ABB RAPID module: 00A6084E

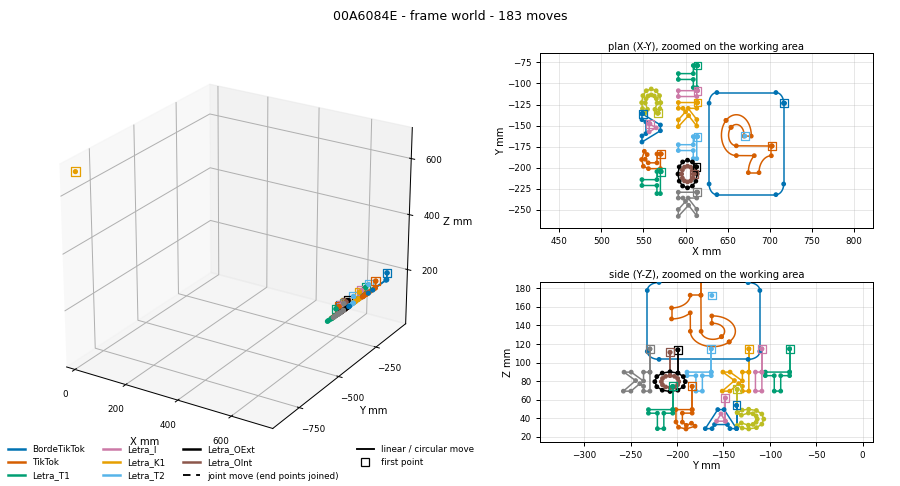
[picture p0: tool path of 00A6084E in frame world, 183 of 183 moves have a stored position in this frame; points joined in program order, loops and branches not executed]
MODULE Module1
        CONST robtarget Target_130_BordeTikTokInicio:=[[92.878,251.287,20],[0.27059805,-0.653281482,0.653281482,0.27059805],[-1,0,-1,0],[9E+09,9E+09,9E+09,9E+09,9E+09,9E+09]];
    CONST robtarget Target_140:=[[83.933,247.582,20],[0.27059805,-0.653281482,0.653281482,0.27059805],[-1,0,-1,0],[9E+09,9E+09,9E+09,9E+09,9E+09,9E+09]];
    CONST robtarget Target_150:=[[80.227,238.636,20],[0.27059805,-0.653281482,0.653281482,0.27059805],[-1,0,-1,0],[9E+09,9E+09,9E+09,9E+09,9E+09,9E+09]];
    CONST robtarget Target_160:=[[80.227,142.704,20],[0.27059805,-0.653281482,0.653281482,0.27059805],[-1,0,-1,0],[9E+09,9E+09,9E+09,9E+09,9E+09,9E+09]];
    CONST robtarget Target_170:=[[83.933,133.759,20],[0.27059805,-0.653281482,0.653281482,0.27059805],[-1,0,-1,0],[9E+09,9E+09,9E+09,9E+09,9E+09,9E+09]];
    CONST robtarget Target_180:=[[92.878,130.054,20],[0.27059805,-0.653281482,0.653281482,0.27059805],[-1,0,-1,0],[9E+09,9E+09,9E+09,9E+09,9E+09,9E+09]];
    CONST robtarget Target_190:=[[188.81,130.054,20],[0.27059805,-0.653281482,0.653281482,0.27059805],[-1,0,-1,0],[9E+09,9E+09,9E+09,9E+09,9E+09,9E+09]];
    CONST robtarget Target_200:=[[197.755,133.759,20],[0.27059805,-0.653281482,0.653281482,0.27059805],[-1,0,-1,0],[9E+09,9E+09,9E+09,9E+09,9E+09,9E+09]];
    CONST robtarget Target_210:=[[201.46,142.704,20],[0.27059805,-0.653281482,0.653281482,0.27059805],[-1,0,-1,0],[9E+09,9E+09,9E+09,9E+09,9E+09,9E+09]];
    CONST robtarget Target_220:=[[201.46,238.636,20],[0.27059805,-0.653281482,0.653281482,0.27059805],[-1,0,-1,0],[9E+09,9E+09,9E+09,9E+09,9E+09,9E+09]];
    CONST robtarget Target_230:=[[197.755,247.582,20],[0.27059805,-0.653281482,0.653281482,0.27059805],[-1,0,-1,0],[9E+09,9E+09,9E+09,9E+09,9E+09,9E+09]];
    CONST robtarget Target_240_BordeTikTokFinal:=[[188.81,251.287,20],[0.27059805,-0.653281482,0.653281482,0.27059805],[-1,0,-1,0],[9E+09,9E+09,9E+09,9E+09,9E+09,9E+09]];
    CONST robtarget Target_250_TikTokInicio:=[[143.706205367,231.257091716,20.000126522],[0.27059805,-0.653281482,0.653281482,0.27059805],[0,0,0,0],[9E+09,9E+09,9E+09,9E+09,9E+09,9E+09]];
    CONST robtarget Target_260:=[[143.479220622,174.279999139,20.000159098],[0.27059805,-0.653281482,0.653281482,0.27059805],[0,0,0,0],[9E+09,9E+09,9E+09,9E+09,9E+09,9E+09]];
    CONST robtarget Target_270:=[[135.378239234,162.526330146,20.000165817],[0.27059805,-0.653281482,0.653281482,0.27059805],[0,0,0,0],[9E+09,9E+09,9E+09,9E+09,9E+09,9E+09]];
    CONST robtarget Target_280:=[[121.484474213,165.803207899,20.000163944],[0.27059805,-0.653281482,0.653281482,0.27059805],[0,0,0,0],[9E+09,9E+09,9E+09,9E+09,9E+09,9E+09]];
    CONST robtarget Target_290:=[[119.489363555,179.938064379,20.000155863],[0.27059805,-0.653281482,0.653281482,0.27059805],[0,0,0,0],[9E+09,9E+09,9E+09,9E+09,9E+09,9E+09]];
    CONST robtarget Target_300:=[[131.933354464,186.932471038,20.000151864],[0.27059805,-0.653281482,0.653281482,0.27059805],[0,0,0,0],[9E+09,9E+09,9E+09,9E+09,9E+09,9E+09]];
    CONST robtarget Target_310:=[[131.979634785,198.549631032,20.000145222],[0.27059805,-0.653281482,0.653281482,0.27059805],[0,0,0,0],[9E+09,9E+09,9E+09,9E+09,9E+09,9E+09]];
    CONST robtarget Target_320:=[[108.772618252,184.400845477,20.000153312],[0.27059805,-0.653281482,0.653281482,0.27059805],[0,0,0,0],[9E+09,9E+09,9E+09,9E+09,9E+09,9E+09]];
    CONST robtarget Target_330:=[[113.281741814,157.597458494,20.000168635],[0.27059805,-0.653281482,0.653281482,0.27059805],[0,0,0,0],[9E+09,9E+09,9E+09,9E+09,9E+09,9E+09]];
    CONST robtarget Target_340:=[[139.840807855,151.820802015,20.000171938],[0.27059805,-0.653281482,0.653281482,0.27059805],[0,0,0,0],[9E+09,9E+09,9E+09,9E+09,9E+09,9E+09]];
    CONST robtarget Target_350:=[[155.075499923,174.329864782,20.000159069],[0.27059805,-0.653281482,0.653281482,0.27059805],[0,0,0,0],[9E+09,9E+09,9E+09,9E+09,9E+09,9E+09]];
    CONST robtarget Target_360:=[[155.17372753,203.510585817,20.000142385],[0.27059805,-0.653281482,0.653281482,0.27059805],[0,0,0,0],[9E+09,9E+09,9E+09,9E+09,9E+09,9E+09]];
    CONST robtarget Target_370:=[[167.73702862,194.971199808,20.000147268],[0.27059805,-0.653281482,0.653281482,0.27059805],[0,0,0,0],[9E+09,9E+09,9E+09,9E+09,9E+09,9E+09]];
    CONST robtarget Target_380:=[[175.332383248,193.829143916,20.000147921],[0.27059805,-0.653281482,0.653281482,0.27059805],[0,0,0,0],[9E+09,9E+09,9E+09,9E+09,9E+09,9E+09]];
    CONST robtarget Target_390:=[[175.332383248,211.188020458,20.000137996],[0.27059805,-0.653281482,0.653281482,0.27059805],[0,0,0,0],[9E+09,9E+09,9E+09,9E+09,9E+09,9E+09]];
    CONST robtarget Target_400:=[[161.14267515,217.065945812,20.00013646],[0.27059805,-0.653281482,0.653281482,0.27059805],[0,0,0,0],[9E+09,9E+09,9E+09,9E+09,9E+09,9E+09]];
    CONST robtarget Target_410_TikTokFinal:=[[155.26722819,231.257091716,20.000126522],[0.27059805,-0.653281482,0.653281482,0.27059805],[0,0,0,0],[9E+09,9E+09,9E+09,9E+09,9E+09,9E+09]];
    CONST robtarget Target_415_T1Inicio:=[[48.177,110.059,20],[0.27059805,-0.653281482,0.653281482,0.27059805],[-1,1,-2,0],[9E+09,9E+09,9E+09,9E+09,9E+09,9E+09]];
    CONST robtarget Target_420:=[[48.174,104.402,20],[0.27059805,-0.653281482,0.653281482,0.27059805],[-1,1,-2,0],[9E+09,9E+09,9E+09,9E+09,9E+09,9E+09]];
    CONST robtarget Target_430:=[[57.774,104.396,20],[0.27059805,-0.653281482,0.653281482,0.27059805],[-1,1,-2,0],[9E+09,9E+09,9E+09,9E+09,9E+09,9E+09]];
    CONST robtarget Target_440:=[[57.759,80.053,20],[0.27059805,-0.653281482,0.653281482,0.27059805],[-1,1,-2,0],[9E+09,9E+09,9E+09,9E+09,9E+09,9E+09]];
    CONST robtarget Target_450:=[[64.701,80.049,20],[0.27059805,-0.653281482,0.653281482,0.27059805],[-1,1,-2,0],[9E+09,9E+09,9E+09,9E+09,9E+09,9E+09]];
    CONST robtarget Target_460:=[[64.717,104.392,20],[0.27059805,-0.653281482,0.653281482,0.27059805],[-1,1,-2,0],[9E+09,9E+09,9E+09,9E+09,9E+09,9E+09]];
    CONST robtarget Target_470:=[[74.317,104.386,20],[0.27059805,-0.653281482,0.653281482,0.27059805],[-1,1,-2,0],[9E+09,9E+09,9E+09,9E+09,9E+09,9E+09]];
    CONST robtarget Target_480_T1Final:=[[74.32,110.043,20],[0.27059805,-0.653281482,0.653281482,0.27059805],[-1,1,-2,0],[9E+09,9E+09,9E+09,9E+09,9E+09,9E+09]];
    CONST robtarget Target_490_IInicio:=[[78.049,110.041,20],[0.27059805,-0.653281482,0.653281482,0.27059805],[-1,1,-2,0],[9E+09,9E+09,9E+09,9E+09,9E+09,9E+09]];
    CONST robtarget Target_500:=[[78.03,80.041,20],[0.27059805,-0.653281482,0.653281482,0.27059805],[-1,1,-2,0],[9E+09,9E+09,9E+09,9E+09,9E+09,9E+09]];
    CONST robtarget Target_510:=[[84.973,80.036,20],[0.27059805,-0.653281482,0.653281482,0.27059805],[-1,1,-2,0],[9E+09,9E+09,9E+09,9E+09,9E+09,9E+09]];
    CONST robtarget Target_520_IFinal:=[[84.992,110.036,20],[0.27059805,-0.653281482,0.653281482,0.27059805],[-1,1,-2,0],[9E+09,9E+09,9E+09,9E+09,9E+09,9E+09]];
    CONST robtarget Target_530_K1Inicio:=[[92.106,110.032,20],[0.27059805,-0.653281482,0.653281482,0.27059805],[-1,1,-2,0],[9E+09,9E+09,9E+09,9E+09,9E+09,9E+09]];
    CONST robtarget Target_540:=[[92.087,80.032,20],[0.27059805,-0.653281482,0.653281482,0.27059805],[-1,1,-2,0],[9E+09,9E+09,9E+09,9E+09,9E+09,9E+09]];
    CONST robtarget Target_550:=[[98.987,80.028,20],[0.27059805,-0.653281482,0.653281482,0.27059805],[-1,1,-2,0],[9E+09,9E+09,9E+09,9E+09,9E+09,9E+09]];
    CONST robtarget Target_560:=[[98.992,87.613,20],[0.27059805,-0.653281482,0.653281482,0.27059805],[-1,1,-2,0],[9E+09,9E+09,9E+09,9E+09,9E+09,9E+09]];
    CONST robtarget Target_570:=[[103.023,91.811,20],[0.27059805,-0.653281482,0.653281482,0.27059805],[-1,1,-2,0],[9E+09,9E+09,9E+09,9E+09,9E+09,9E+09]];
    CONST robtarget Target_580:=[[112.616,80.019,20],[0.27059805,-0.653281482,0.653281482,0.27059805],[-1,1,-2,0],[9E+09,9E+09,9E+09,9E+09,9E+09,9E+09]];
    CONST robtarget Target_590:=[[120.716,80.014,20],[0.27059805,-0.653281482,0.653281482,0.27059805],[-1,1,-2,0],[9E+09,9E+09,9E+09,9E+09,9E+09,9E+09]];
    CONST robtarget Target_600:=[[107.569,96.651,20],[0.27059805,-0.653281482,0.653281482,0.27059805],[-1,1,-2,0],[9E+09,9E+09,9E+09,9E+09,9E+09,9E+09]];
    CONST robtarget Target_610:=[[120.006,110.015,20],[0.27059805,-0.653281482,0.653281482,0.27059805],[-1,0,-2,0],[9E+09,9E+09,9E+09,9E+09,9E+09,9E+09]];
    CONST robtarget Target_620:=[[112.292,110.019,20],[0.27059805,-0.653281482,0.653281482,0.27059805],[-1,1,-2,0],[9E+09,9E+09,9E+09,9E+09,9E+09,9E+09]];
    CONST robtarget Target_630:=[[98.997,96.013,20],[0.27059805,-0.653281482,0.653281482,0.27059805],[-1,1,-2,0],[9E+09,9E+09,9E+09,9E+09,9E+09,9E+09]];
    CONST robtarget Target_640_K1Final:=[[99.006,110.028,20],[0.27059805,-0.653281482,0.653281482,0.27059805],[-1,1,-2,0],[9E+09,9E+09,9E+09,9E+09,9E+09,9E+09]];
    CONST robtarget Target_650_T2Inicio:=[[132.563,110.007,20],[0.27059805,-0.653281482,0.653281482,0.27059805],[0,0,0,0],[9E+09,9E+09,9E+09,9E+09,9E+09,9E+09]];
    CONST robtarget Target_660:=[[132.559,104.35,20],[0.27059805,-0.653281482,0.653281482,0.27059805],[-1,1,-2,0],[9E+09,9E+09,9E+09,9E+09,9E+09,9E+09]];
    CONST robtarget Target_670:=[[142.159,104.344,20],[0.27059805,-0.653281482,0.653281482,0.27059805],[-1,0,-2,0],[9E+09,9E+09,9E+09,9E+09,9E+09,9E+09]];
    CONST robtarget Target_680:=[[142.144,80.001,20],[0.27059805,-0.653281482,0.653281482,0.27059805],[-1,1,-2,0],[9E+09,9E+09,9E+09,9E+09,9E+09,9E+09]];
    CONST robtarget Target_690:=[[149.087,79.996,20],[0.27059805,-0.653281482,0.653281482,0.27059805],[-1,1,-2,0],[9E+09,9E+09,9E+09,9E+09,9E+09,9E+09]];
    CONST robtarget Target_700:=[[149.102,104.339,20],[0.27059805,-0.653281482,0.653281482,0.27059805],[-1,0,-2,0],[9E+09,9E+09,9E+09,9E+09,9E+09,9E+09]];
    CONST robtarget Target_710:=[[158.702,104.333,20],[0.27059805,-0.653281482,0.653281482,0.27059805],[-1,0,-2,0],[9E+09,9E+09,9E+09,9E+09,9E+09,9E+09]];
    CONST robtarget Target_720_T2Final:=[[158.706,109.99,20],[0.27059805,-0.653281482,0.653281482,0.27059805],[-1,0,-2,0],[9E+09,9E+09,9E+09,9E+09,9E+09,9E+09]];
    CONST robtarget Target_730_OExtInicio:=[[168.541,108.484,20],[0.27059805,-0.653281482,0.653281482,0.27059805],[0,0,0,0],[9E+09,9E+09,9E+09,9E+09,9E+09,9E+09]];
    CONST robtarget Target_740:=[[162.666,102.938,20],[0.27059805,-0.653281482,0.653281482,0.27059805],[-1,0,-2,0],[9E+09,9E+09,9E+09,9E+09,9E+09,9E+09]];
    CONST robtarget Target_750:=[[160.539,94.989,20],[0.27059805,-0.653281482,0.653281482,0.27059805],[-1,1,-2,0],[9E+09,9E+09,9E+09,9E+09,9E+09,9E+09]];
    CONST robtarget Target_760:=[[162.656,87.038,20],[0.27059805,-0.653281482,0.653281482,0.27059805],[-1,1,-2,0],[9E+09,9E+09,9E+09,9E+09,9E+09,9E+09]];
    CONST robtarget Target_770:=[[168.524,81.484,20],[0.27059805,-0.653281482,0.653281482,0.27059805],[-1,1,-2,0],[9E+09,9E+09,9E+09,9E+09,9E+09,9E+09]];
    CONST robtarget Target_780:=[[176.944,79.465,20],[0.27059805,-0.653281482,0.653281482,0.27059805],[-1,1,-2,0],[9E+09,9E+09,9E+09,9E+09,9E+09,9E+09]];
    CONST robtarget Target_790:=[[185.345,81.474,20],[0.27059805,-0.653281482,0.653281482,0.27059805],[-1,1,-2,0],[9E+09,9E+09,9E+09,9E+09,9E+09,9E+09]];
    CONST robtarget Target_800:=[[191.22,87.02,20],[0.27059805,-0.653281482,0.653281482,0.27059805],[-1,0,-2,0],[9E+09,9E+09,9E+09,9E+09,9E+09,9E+09]];
    CONST robtarget Target_810:=[[193.368,94.969,20],[0.27059805,-0.653281482,0.653281482,0.27059805],[-1,0,-2,0],[9E+09,9E+09,9E+09,9E+09,9E+09,9E+09]];
    CONST robtarget Target_820:=[[191.23,102.92,20],[0.27059805,-0.653281482,0.653281482,0.27059805],[-1,0,-2,0],[9E+09,9E+09,9E+09,9E+09,9E+09,9E+09]];
    CONST robtarget Target_830:=[[185.362,108.474,20],[0.27059805,-0.653281482,0.653281482,0.27059805],[-1,0,-2,0],[9E+09,9E+09,9E+09,9E+09,9E+09,9E+09]];
    CONST robtarget Target_840_OExtFinal:=[[176.963,110.493,20],[0.27059805,-0.653281482,0.653281482,0.27059805],[-1,0,-2,0],[9E+09,9E+09,9E+09,9E+09,9E+09,9E+09]];
    CONST robtarget Target_850_OIntInicio:=[[176.96,104.579,20],[0.27059805,-0.653281482,0.653281482,0.27059805],[0,0,0,0],[9E+09,9E+09,9E+09,9E+09,9E+09,9E+09]];
    CONST robtarget Target_860:=[[172.159,103.361,20],[0.27059805,-0.653281482,0.653281482,0.27059805],[-1,0,-2,0],[9E+09,9E+09,9E+09,9E+09,9E+09,9E+09]];
    CONST robtarget Target_870:=[[168.792,99.956,20],[0.27059805,-0.653281482,0.653281482,0.27059805],[-1,0,-2,0],[9E+09,9E+09,9E+09,9E+09,9E+09,9E+09]];
    CONST robtarget Target_880:=[[167.568,94.985,20],[0.27059805,-0.653281482,0.653281482,0.27059805],[-1,0,-2,0],[9E+09,9E+09,9E+09,9E+09,9E+09,9E+09]];
    CONST robtarget Target_890:=[[168.786,90.013,20],[0.27059805,-0.653281482,0.653281482,0.27059805],[-1,1,-2,0],[9E+09,9E+09,9E+09,9E+09,9E+09,9E+09]];
    CONST robtarget Target_900:=[[172.148,86.603,20],[0.27059805,-0.653281482,0.653281482,0.27059805],[-1,1,-2,0],[9E+09,9E+09,9E+09,9E+09,9E+09,9E+09]];
    CONST robtarget Target_910:=[[176.948,85.379,20],[0.27059805,-0.653281482,0.653281482,0.27059805],[-1,1,-2,0],[9E+09,9E+09,9E+09,9E+09,9E+09,9E+09]];
    CONST robtarget Target_920:=[[181.748,86.597,20],[0.27059805,-0.653281482,0.653281482,0.27059805],[-1,1,-2,0],[9E+09,9E+09,9E+09,9E+09,9E+09,9E+09]];
    CONST robtarget Target_930:=[[185.115,90.003,20],[0.27059805,-0.653281482,0.653281482,0.27059805],[-1,0,-2,0],[9E+09,9E+09,9E+09,9E+09,9E+09,9E+09]];
    CONST robtarget Target_940:=[[186.339,94.973,20],[0.27059805,-0.653281482,0.653281482,0.27059805],[-1,0,-2,0],[9E+09,9E+09,9E+09,9E+09,9E+09,9E+09]];
    CONST robtarget Target_950:=[[185.121,99.945,20],[0.27059805,-0.653281482,0.653281482,0.27059805],[-1,0,-2,0],[9E+09,9E+09,9E+09,9E+09,9E+09,9E+09]];
    CONST robtarget Target_960_OIntFinal:=[[181.759,103.355,20],[0.27059805,-0.653281482,0.653281482,0.27059805],[-1,0,-2,0],[9E+09,9E+09,9E+09,9E+09,9E+09,9E+09]];
    CONST robtarget Target_970_K2Inicio:=[[198.606,109.966,20],[0.27059805,-0.653281482,0.653281482,0.27059805],[0,0,0,0],[9E+09,9E+09,9E+09,9E+09,9E+09,9E+09]];
    CONST robtarget Target_980:=[[198.587,79.966,20],[0.27059805,-0.653281482,0.653281482,0.27059805],[-1,1,-2,0],[9E+09,9E+09,9E+09,9E+09,9E+09,9E+09]];
    CONST robtarget Target_990:=[[205.487,79.961,20],[0.27059805,-0.653281482,0.653281482,0.27059805],[-1,0,-2,0],[9E+09,9E+09,9E+09,9E+09,9E+09,9E+09]];
    CONST robtarget Target_1000:=[[205.492,87.547,20],[0.27059805,-0.653281482,0.653281482,0.27059805],[-1,0,-2,0],[9E+09,9E+09,9E+09,9E+09,9E+09,9E+09]];
    CONST robtarget Target_1010:=[[209.523,91.744,20],[0.27059805,-0.653281482,0.653281482,0.27059805],[-1,0,-2,0],[9E+09,9E+09,9E+09,9E+09,9E+09,9E+09]];
    CONST robtarget Target_1020:=[[219.116,79.953,20],[0.27059805,-0.653281482,0.653281482,0.27059805],[-1,0,-2,0],[9E+09,9E+09,9E+09,9E+09,9E+09,9E+09]];
    CONST robtarget Target_1030:=[[227.216,79.948,20],[0.27059805,-0.653281482,0.653281482,0.27059805],[-1,0,-2,0],[9E+09,9E+09,9E+09,9E+09,9E+09,9E+09]];
    CONST robtarget Target_1040:=[[214.069,96.584,20],[0.27059805,-0.653281482,0.653281482,0.27059805],[-1,0,-2,0],[9E+09,9E+09,9E+09,9E+09,9E+09,9E+09]];
    CONST robtarget Target_1050:=[[226.506,109.948,20],[0.27059805,-0.653281482,0.653281482,0.27059805],[-1,0,-1,0],[9E+09,9E+09,9E+09,9E+09,9E+09,9E+09]];
    CONST robtarget Target_1060:=[[218.792,109.953,20],[0.27059805,-0.653281482,0.653281482,0.27059805],[-1,0,-2,0],[9E+09,9E+09,9E+09,9E+09,9E+09,9E+09]];
    CONST robtarget Target_1070:=[[205.497,95.947,20],[0.27059805,-0.653281482,0.653281482,0.27059805],[-1,0,-2,0],[9E+09,9E+09,9E+09,9E+09,9E+09,9E+09]];
    CONST robtarget Target_1080_K2Final:=[[205.506,109.961,20],[0.27059805,-0.653281482,0.653281482,0.27059805],[-1,0,-2,0],[9E+09,9E+09,9E+09,9E+09,9E+09,9E+09]];
    CONST robtarget Target_1090_CInicio:=[[104.623,46.124,20],[0.27059805,-0.653281482,0.653281482,0.27059805],[-1,1,-2,0],[9E+09,9E+09,9E+09,9E+09,9E+09,9E+09]];
    CONST robtarget Target_1100:=[[99.333,50.07,20],[0.27059805,-0.653281482,0.653281482,0.27059805],[-1,1,-2,0],[9E+09,9E+09,9E+09,9E+09,9E+09,9E+09]];
    CONST robtarget Target_1110:=[[92.284,51.446,20],[0.27059805,-0.653281482,0.653281482,0.27059805],[-1,1,-2,0],[9E+09,9E+09,9E+09,9E+09,9E+09,9E+09]];
    CONST robtarget Target_1120:=[[83.947,49.459,20],[0.27059805,-0.653281482,0.653281482,0.27059805],[-1,1,-2,0],[9E+09,9E+09,9E+09,9E+09,9E+09,9E+09]];
    CONST robtarget Target_1130:=[[78.115,43.934,20],[0.27059805,-0.653281482,0.653281482,0.27059805],[-1,1,-2,0],[9E+09,9E+09,9E+09,9E+09,9E+09,9E+09]];
    CONST robtarget Target_1140:=[[75.988,35.942,20],[0.27059805,-0.653281482,0.653281482,0.27059805],[-1,1,-2,0],[9E+09,9E+09,9E+09,9E+09,9E+09,9E+09]];
    CONST robtarget Target_1150:=[[78.105,27.948,20],[0.27059805,-0.653281482,0.653281482,0.27059805],[-1,1,-2,0],[9E+09,9E+09,9E+09,9E+09,9E+09,9E+09]];
    CONST robtarget Target_1160:=[[83.93,22.416,20],[0.27059805,-0.653281482,0.653281482,0.27059805],[-1,1,-2,0],[9E+09,9E+09,9E+09,9E+09,9E+09,9E+09]];
    CONST robtarget Target_1170:=[[92.221,20.418,20],[0.27059805,-0.653281482,0.653281482,0.27059805],[-1,1,-2,0],[9E+09,9E+09,9E+09,9E+09,9E+09,9E+09]];
    CONST robtarget Target_1180:=[[99.294,21.785,20],[0.27059805,-0.653281482,0.653281482,0.27059805],[-1,1,-2,0],[9E+09,9E+09,9E+09,9E+09,9E+09,9E+09]];
    CONST robtarget Target_1190:=[[104.61,25.767,20],[0.27059805,-0.653281482,0.653281482,0.27059805],[-1,1,-2,0],[9E+09,9E+09,9E+09,9E+09,9E+09,9E+09]];
    CONST robtarget Target_1200:=[[100.156,29.884,20],[0.27059805,-0.653281482,0.653281482,0.27059805],[-1,1,-2,0],[9E+09,9E+09,9E+09,9E+09,9E+09,9E+09]];
    CONST robtarget Target_1210:=[[92.611,26.332,20],[0.27059805,-0.653281482,0.653281482,0.27059805],[-1,1,-2,0],[9E+09,9E+09,9E+09,9E+09,9E+09,9E+09]];
    CONST robtarget Target_1220:=[[87.64,27.556,20],[0.27059805,-0.653281482,0.653281482,0.27059805],[-1,1,-2,0],[9E+09,9E+09,9E+09,9E+09,9E+09,9E+09]];
    CONST robtarget Target_1230:=[[84.235,30.965,20],[0.27059805,-0.653281482,0.653281482,0.27059805],[-1,1,-2,0],[9E+09,9E+09,9E+09,9E+09,9E+09,9E+09]];
    CONST robtarget Target_1240:=[[83.017,35.938,20],[0.27059805,-0.653281482,0.653281482,0.27059805],[-1,1,-2,0],[9E+09,9E+09,9E+09,9E+09,9E+09,9E+09]];
    CONST robtarget Target_1250:=[[84.241,40.908,20],[0.27059805,-0.653281482,0.653281482,0.27059805],[-1,1,-2,0],[9E+09,9E+09,9E+09,9E+09,9E+09,9E+09]];
    CONST robtarget Target_1260:=[[87.651,44.313,20],[0.27059805,-0.653281482,0.653281482,0.27059805],[-1,1,-2,0],[9E+09,9E+09,9E+09,9E+09,9E+09,9E+09]];
    CONST robtarget Target_1270:=[[92.623,45.532,20],[0.27059805,-0.653281482,0.653281482,0.27059805],[-1,1,-2,0],[9E+09,9E+09,9E+09,9E+09,9E+09,9E+09]];
    CONST robtarget Target_1280_CFinal:=[[100.163,42.013,20],[0.27059805,-0.653281482,0.653281482,0.27059805],[-1,1,-2,0],[9E+09,9E+09,9E+09,9E+09,9E+09,9E+09]];
    CONST robtarget Target_1290_AExtInicio:=[[105.336,20.924,20],[0.27059805,-0.653281482,0.653281482,0.27059805],[-1,1,-2,0],[9E+09,9E+09,9E+09,9E+09,9E+09,9E+09]];
    CONST robtarget Target_1300:=[[118.726,50.915,20],[0.27059805,-0.653281482,0.653281482,0.27059805],[-1,1,-2,0],[9E+09,9E+09,9E+09,9E+09,9E+09,9E+09]];
    CONST robtarget Target_1310:=[[125.583,50.911,20],[0.27059805,-0.653281482,0.653281482,0.27059805],[-1,1,-2,0],[9E+09,9E+09,9E+09,9E+09,9E+09,9E+09]];
    CONST robtarget Target_1320:=[[138.979,20.903,20],[0.27059805,-0.653281482,0.653281482,0.27059805],[-1,1,-2,0],[9E+09,9E+09,9E+09,9E+09,9E+09,9E+09]];
    CONST robtarget Target_1330:=[[131.693,20.907,20],[0.27059805,-0.653281482,0.653281482,0.27059805],[-1,1,-2,0],[9E+09,9E+09,9E+09,9E+09,9E+09,9E+09]];
    CONST robtarget Target_1340:=[[129.04,27.338,20],[0.27059805,-0.653281482,0.653281482,0.27059805],[-1,1,-2,0],[9E+09,9E+09,9E+09,9E+09,9E+09,9E+09]];
    CONST robtarget Target_1350:=[[115.111,27.346,20],[0.27059805,-0.653281482,0.653281482,0.27059805],[-1,1,-2,0],[9E+09,9E+09,9E+09,9E+09,9E+09,9E+09]];
    CONST robtarget Target_1360_AExtFinal:=[[112.45,20.919,20],[0.27059805,-0.653281482,0.653281482,0.27059805],[-1,1,-2,0],[9E+09,9E+09,9E+09,9E+09,9E+09,9E+09]];
    CONST robtarget Target_1400_JInicio:=[[153.14,50.894,20],[0.27059805,-0.653281482,0.653281482,0.27059805],[-1,1,-2,0],[9E+09,9E+09,9E+09,9E+09,9E+09,9E+09]];
    CONST robtarget Target_1410:=[[153.137,45.322,20],[0.27059805,-0.653281482,0.653281482,0.27059805],[-1,1,-2,0],[9E+09,9E+09,9E+09,9E+09,9E+09,9E+09]];
    CONST robtarget Target_1420:=[[163.68,45.316,20],[0.27059805,-0.653281482,0.653281482,0.27059805],[-1,1,-2,0],[9E+09,9E+09,9E+09,9E+09,9E+09,9E+09]];
    CONST robtarget Target_1430:=[[163.671,31.044,20],[0.27059805,-0.653281482,0.653281482,0.27059805],[-1,1,-2,0],[9E+09,9E+09,9E+09,9E+09,9E+09,9E+09]];
    CONST robtarget Target_1440:=[[159.425,26.076,20],[0.27059805,-0.653281482,0.653281482,0.27059805],[-1,1,-2,0],[9E+09,9E+09,9E+09,9E+09,9E+09,9E+09]];
    CONST robtarget Target_1450:=[[153.856,29.379,20],[0.27059805,-0.653281482,0.653281482,0.27059805],[-1,1,-2,0],[9E+09,9E+09,9E+09,9E+09,9E+09,9E+09]];
    CONST robtarget Target_1460:=[[149.996,24.753,20],[0.27059805,-0.653281482,0.653281482,0.27059805],[-1,1,-2,0],[9E+09,9E+09,9E+09,9E+09,9E+09,9E+09]];
    CONST robtarget Target_1470:=[[159.764,20.375,20],[0.27059805,-0.653281482,0.653281482,0.27059805],[-1,1,-2,0],[9E+09,9E+09,9E+09,9E+09,9E+09,9E+09]];
    CONST robtarget Target_1480:=[[167.823,23.135,20],[0.27059805,-0.653281482,0.653281482,0.27059805],[-1,1,-2,0],[9E+09,9E+09,9E+09,9E+09,9E+09,9E+09]];
    CONST robtarget Target_1490:=[[170.571,31.426,20],[0.27059805,-0.653281482,0.653281482,0.27059805],[-1,1,-2,0],[9E+09,9E+09,9E+09,9E+09,9E+09,9E+09]];
    CONST robtarget Target_1500_JFinal:=[[170.583,50.883,20],[0.27059805,-0.653281482,0.653281482,0.27059805],[-1,1,-2,0],[9E+09,9E+09,9E+09,9E+09,9E+09,9E+09]];
    CONST robtarget Target_1510_T3Inicio:=[[174.055,50.881,20],[0.27059805,-0.653281482,0.653281482,0.27059805],[-1,1,-2,0],[9E+09,9E+09,9E+09,9E+09,9E+09,9E+09]];
    CONST robtarget Target_1520:=[[174.051,45.224,20],[0.27059805,-0.653281482,0.653281482,0.27059805],[-1,1,-2,0],[9E+09,9E+09,9E+09,9E+09,9E+09,9E+09]];
    CONST robtarget Target_1530:=[[183.651,45.218,20],[0.27059805,-0.653281482,0.653281482,0.27059805],[-1,1,-2,0],[9E+09,9E+09,9E+09,9E+09,9E+09,9E+09]];
    CONST robtarget Target_1540:=[[183.636,20.875,20],[0.27059805,-0.653281482,0.653281482,0.27059805],[-1,1,-2,0],[9E+09,9E+09,9E+09,9E+09,9E+09,9E+09]];
    CONST robtarget Target_1550:=[[190.579,20.871,20],[0.27059805,-0.653281482,0.653281482,0.27059805],[-1,1,-2,0],[9E+09,9E+09,9E+09,9E+09,9E+09,9E+09]];
    CONST robtarget Target_1560:=[[190.594,45.213,20],[0.27059805,-0.653281482,0.653281482,0.27059805],[-1,1,-2,0],[9E+09,9E+09,9E+09,9E+09,9E+09,9E+09]];
    CONST robtarget Target_1570:=[[200.194,45.207,20],[0.27059805,-0.653281482,0.653281482,0.27059805],[-1,1,-2,0],[9E+09,9E+09,9E+09,9E+09,9E+09,9E+09]];
    CONST robtarget Target_1580_T3Final:=[[200.198,50.865,20],[0.27059805,-0.653281482,0.653281482,0.27059805],[-1,1,-2,0],[9E+09,9E+09,9E+09,9E+09,9E+09,9E+09]];
    CONST robtarget Target_1370_AIntInicio:=[[117.343,32.616,20],[0.27059805,-0.653281482,0.653281482,0.27059805],[-1,1,-2,0],[9E+09,9E+09,9E+09,9E+09,9E+09,9E+09]];
    CONST robtarget Target_1380:=[[122.108,44.099,20],[0.27059805,-0.653281482,0.653281482,0.27059805],[-1,1,-2,0],[9E+09,9E+09,9E+09,9E+09,9E+09,9E+09]];
    CONST robtarget Target_1390_AIntFinal:=[[126.858,32.61,20],[0.27059805,-0.653281482,0.653281482,0.27059805],[-1,1,-2,0],[9E+09,9E+09,9E+09,9E+09,9E+09,9E+09]];
    CONST robtarget Target_130_BordeTikTokInicio_4:=[[92.878,268.964669525,37.677669535],[0.27059805,-0.653281482,0.653281482,0.27059805],[-1,0,-1,0],[9E+09,9E+09,9E+09,9E+09,9E+09,9E+09]];
    CONST robtarget Target_250_TikTokInicio_2:=[[143.706205367,248.934761241,37.677796057],[0.27059805,-0.653281482,0.653281482,0.27059805],[-1,0,-1,0],[9E+09,9E+09,9E+09,9E+09,9E+09,9E+09]];
    CONST robtarget Target_415_T1Inicio_2:=[[48.177,127.736669525,37.677669535],[0.27059805,-0.653281482,0.653281482,0.27059805],[-1,0,-1,0],[9E+09,9E+09,9E+09,9E+09,9E+09,9E+09]];
    CONST robtarget Target_490_IInicio_2:=[[78.049,127.718669525,37.677669535],[0.27059805,-0.653281482,0.653281482,0.27059805],[-1,0,-1,0],[9E+09,9E+09,9E+09,9E+09,9E+09,9E+09]];
    CONST robtarget Target_530_K1Inicio_2:=[[92.106,127.709669525,37.677669535],[0.27059805,-0.653281482,0.653281482,0.27059805],[-1,0,-1,0],[9E+09,9E+09,9E+09,9E+09,9E+09,9E+09]];
    CONST robtarget Target_650_T2Inicio_2:=[[132.563,127.684669525,37.677669535],[0.27059805,-0.653281482,0.653281482,0.27059805],[-1,0,-1,0],[9E+09,9E+09,9E+09,9E+09,9E+09,9E+09]];
    CONST robtarget Target_730_OExtInicio_2:=[[168.541,126.161669525,37.677669535],[0.27059805,-0.653281482,0.653281482,0.27059805],[-1,0,-1,0],[9E+09,9E+09,9E+09,9E+09,9E+09,9E+09]];
    CONST robtarget Target_850_OIntInicio_3:=[[176.96,122.256669525,37.677669535],[0.27059805,-0.653281482,0.653281482,0.27059805],[-1,0,-1,0],[9E+09,9E+09,9E+09,9E+09,9E+09,9E+09]];
    CONST robtarget Target_970_K2Inicio_2:=[[198.606,127.643669525,37.677669535],[0.27059805,-0.653281482,0.653281482,0.27059805],[-1,0,-1,0],[9E+09,9E+09,9E+09,9E+09,9E+09,9E+09]];
    CONST robtarget Target_1090_CInicio_2:=[[104.623,63.801669525,37.677669535],[0.27059805,-0.653281482,0.653281482,0.27059805],[-1,1,-2,0],[9E+09,9E+09,9E+09,9E+09,9E+09,9E+09]];
    CONST robtarget Target_1290_AExtInicio_2:=[[105.336,38.601669525,37.677669535],[0.27059805,-0.653281482,0.653281482,0.27059805],[-1,1,-2,0],[9E+09,9E+09,9E+09,9E+09,9E+09,9E+09]];
    CONST robtarget Target_1400_JInicio_2:=[[153.14,68.571669525,37.677669535],[0.27059805,-0.653281482,0.653281482,0.27059805],[-1,1,-2,0],[9E+09,9E+09,9E+09,9E+09,9E+09,9E+09]];
    CONST robtarget Target_1510_T3Inicio_2:=[[174.055,68.558669525,37.677669535],[0.27059805,-0.653281482,0.653281482,0.27059805],[-1,1,-2,0],[9E+09,9E+09,9E+09,9E+09,9E+09,9E+09]];
    CONST robtarget Target_1370_AIntInicio_2:=[[117.343,50.293669525,37.677669535],[0.27059805,-0.653281482,0.653281482,0.27059805],[-1,1,-2,0],[9E+09,9E+09,9E+09,9E+09,9E+09,9E+09]];
    CONST robtarget PosMantenimiento:=[[842.764,64.247888054,868.878653416],[0.859297836,-0.339353237,0.355932818,-0.140564712],[-2,0,-1,0],[9E+09,9E+09,9E+09,9E+09,9E+09,9E+09]];
    PERS tooldata MyNewTool:=[TRUE,[[120.323,-0.111,166.727],[0.923879533,0,-0.382683432,0]],[1,[0,0,1],[1,0,0,0],0,0,0]];
    TASK PERS wobjdata Workobject_1:=[FALSE,TRUE,"",[[546.66,-30.515,0],[0.657678091,0.259729722,-0.259729722,-0.657678091]],[[0,0,0],[1,0,0,0]]];
    CONST robtarget MyHome:=[[131.933354464,208.145674467,41.213355305],[0.27059805,-0.653281482,0.653281482,0.27059805],[0,0,0,0],[9E+09,9E+09,9E+09,9E+09,9E+09,9E+09]];
!***********************************************************
    !
    ! M?dulo:  Module1
    !
    ! Descripción:
    !   <Introduzca la descripción aquí>
    !
    ! Autor: Cami
    !
    ! Versión: 1.0
    !
    !***********************************************************


    !***********************************************************
    !
    ! Procedimiento Main
    !
    !   Este es el punto de entrada de su programa
    !
    !***********************************************************
    PROC main()
        VAR bool mant := FALSE;

        WHILE TRUE DO

            IF DI_01 = 1 THEN
                SetDO DO_02,1;
                COMPLETO;
                SetDO DO_02,0;
            ENDIF

            IF DI_02 = 1 THEN
                IF mant = FALSE THEN
                    mant := TRUE;
                    Home;
                ELSE
                    mant := FALSE;
                    SetDO DO_02,1;
                    Mantenimiento;
                    SetDO DO_02,0;
                ENDIF

            ENDIF

        ENDWHILE
        SetDO DO_02,0;
        SetDO DO_02,1;
    ENDPROC
    PROC COMPLETO()
        BordeTikTok;
        TikTok;
        Letra_T1;
        Letra_I;
        Letra_K1;
        Letra_T2;
        Letra_OExt;
        Letra_OInt;
        Letra_K2;
        Letra_C;
        Letra_AExt;
        Letra_AInt;
        Letra_J;
        Letra_T3;
    ENDPROC
    PROC BordeTikTok()
        MoveJ Target_130_BordeTikTokInicio_4,v100,z100,MyNewTool\WObj:=Workobject_1;
        MoveJ Target_130_BordeTikTokInicio,v400,z100,MyNewTool\WObj:=Workobject_1;
        MoveC Target_140,Target_150,v100,z100,MyNewTool\WObj:=Workobject_1;
        MoveL Target_160,v100,z100,MyNewTool\WObj:=Workobject_1;
        MoveC Target_170,Target_180,v100,z100,MyNewTool\WObj:=Workobject_1;
        MoveL Target_190,v100,z100,MyNewTool\WObj:=Workobject_1;
        MoveC Target_200,Target_210,v100,z100,MyNewTool\WObj:=Workobject_1;
        MoveL Target_220,v100,z100,MyNewTool\WObj:=Workobject_1;
        MoveC Target_230,Target_240_BordeTikTokFinal,v100,z100,MyNewTool\WObj:=Workobject_1;
        MoveL Target_130_BordeTikTokInicio,v100,z100,MyNewTool\WObj:=Workobject_1;
        MoveL Target_130_BordeTikTokInicio_4,v100,z100,MyNewTool\WObj:=Workobject_1;
    ENDPROC
    PROC TikTok()
        MoveL Target_250_TikTokInicio_2,v100,z100,MyNewTool\WObj:=Workobject_1;
        MoveL Target_250_TikTokInicio,v100,z100,MyNewTool\WObj:=Workobject_1;
        MoveL Target_260,v100,z100,MyNewTool\WObj:=Workobject_1;
        MoveC Target_270,Target_280,v100,z100,MyNewTool\WObj:=Workobject_1;
        MoveL Target_280,v100,z100,MyNewTool\WObj:=Workobject_1;
        MoveC Target_290,Target_300,v100,z100,MyNewTool\WObj:=Workobject_1;
        MoveL Target_310,v100,z100,MyNewTool\WObj:=Workobject_1;
        MoveC Target_320,Target_330,v100,z100,MyNewTool\WObj:=Workobject_1;
        MoveL Target_330,v100,z100,MyNewTool\WObj:=Workobject_1;
        MoveC Target_340,Target_350,v100,z100,MyNewTool\WObj:=Workobject_1;
        MoveL Target_360,v100,z100,MyNewTool\WObj:=Workobject_1;
        MoveC Target_370,Target_380,v100,z100,MyNewTool\WObj:=Workobject_1;
        MoveL Target_390,v100,z100,MyNewTool\WObj:=Workobject_1;
        MoveC Target_400,Target_410_TikTokFinal,v100,z100,MyNewTool\WObj:=Workobject_1;
        MoveL Target_250_TikTokInicio,v100,z100,MyNewTool\WObj:=Workobject_1;
        MoveL Target_250_TikTokInicio_2,v100,z100,MyNewTool\WObj:=Workobject_1;
    ENDPROC
    PROC Letra_T1()
        MoveL Target_415_T1Inicio_2,v100,z100,MyNewTool\WObj:=Workobject_1;
        MoveL Target_415_T1Inicio,v100,z100,MyNewTool\WObj:=Workobject_1;
        MoveL Target_420,v100,z100,MyNewTool\WObj:=Workobject_1;
        MoveL Target_430,v100,z100,MyNewTool\WObj:=Workobject_1;
        MoveL Target_440,v100,z100,MyNewTool\WObj:=Workobject_1;
        MoveL Target_450,v100,z100,MyNewTool\WObj:=Workobject_1;
        MoveL Target_460,v100,z100,MyNewTool\WObj:=Workobject_1;
        MoveL Target_470,v100,z100,MyNewTool\WObj:=Workobject_1;
        MoveL Target_480_T1Final,v100,z100,MyNewTool\WObj:=Workobject_1;
        MoveL Target_415_T1Inicio,v100,z100,MyNewTool\WObj:=Workobject_1;
        MoveL Target_415_T1Inicio_2,v100,z100,MyNewTool\WObj:=Workobject_1;
    ENDPROC
    PROC Letra_I()
        MoveL Target_490_IInicio_2,v100,z100,MyNewTool\WObj:=Workobject_1;
        MoveL Target_490_IInicio,v100,z100,MyNewTool\WObj:=Workobject_1;
        MoveL Target_500,v100,z100,MyNewTool\WObj:=Workobject_1;
        MoveL Target_510,v100,z100,MyNewTool\WObj:=Workobject_1;
        MoveL Target_520_IFinal,v100,z100,MyNewTool\WObj:=Workobject_1;
        MoveL Target_490_IInicio,v100,z100,MyNewTool\WObj:=Workobject_1;
        MoveL Target_490_IInicio_2,v100,z100,MyNewTool\WObj:=Workobject_1;
    ENDPROC
    PROC Letra_K1()
        MoveL Target_530_K1Inicio_2,v100,z100,MyNewTool\WObj:=Workobject_1;
        MoveL Target_530_K1Inicio,v100,z100,MyNewTool\WObj:=Workobject_1;
        MoveL Target_540,v100,z100,MyNewTool\WObj:=Workobject_1;
        MoveL Target_550,v100,z100,MyNewTool\WObj:=Workobject_1;
        MoveL Target_560,v100,z100,MyNewTool\WObj:=Workobject_1;
        MoveL Target_570,v100,z100,MyNewTool\WObj:=Workobject_1;
        MoveL Target_580,v100,z100,MyNewTool\WObj:=Workobject_1;
        MoveL Target_590,v100,z100,MyNewTool\WObj:=Workobject_1;
        MoveL Target_600,v100,z100,MyNewTool\WObj:=Workobject_1;
        MoveL Target_610,v100,z100,MyNewTool\WObj:=Workobject_1;
        MoveL Target_620,v100,z100,MyNewTool\WObj:=Workobject_1;
        MoveL Target_630,v100,z100,MyNewTool\WObj:=Workobject_1;
        MoveL Target_640_K1Final,v100,z100,MyNewTool\WObj:=Workobject_1;
        MoveL Target_530_K1Inicio,v100,z100,MyNewTool\WObj:=Workobject_1;
        MoveL Target_530_K1Inicio_2,v100,z100,MyNewTool\WObj:=Workobject_1;
    ENDPROC
    PROC Letra_T2()
        MoveL Target_650_T2Inicio_2,v100,z100,MyNewTool\WObj:=Workobject_1;
        MoveL Target_650_T2Inicio,v100,z100,MyNewTool\WObj:=Workobject_1;
        MoveL Target_660,v100,z100,MyNewTool\WObj:=Workobject_1;
        MoveL Target_670,v100,z100,MyNewTool\WObj:=Workobject_1;
        MoveL Target_680,v100,z100,MyNewTool\WObj:=Workobject_1;
        MoveL Target_690,v100,z100,MyNewTool\WObj:=Workobject_1;
        MoveL Target_700,v100,z100,MyNewTool\WObj:=Workobject_1;
        MoveL Target_710,v100,z100,MyNewTool\WObj:=Workobject_1;
        MoveL Target_720_T2Final,v100,z100,MyNewTool\WObj:=Workobject_1;
        MoveL Target_650_T2Inicio,v100,z100,MyNewTool\WObj:=Workobject_1;
        MoveL Target_650_T2Inicio_2,v100,z100,MyNewTool\WObj:=Workobject_1;
    ENDPROC
    PROC Letra_OExt()
        MoveL Target_730_OExtInicio_2,v100,z100,MyNewTool\WObj:=Workobject_1;
        MoveL Target_730_OExtInicio,v100,z100,MyNewTool\WObj:=Workobject_1;
        MoveL Target_740,v100,z100,MyNewTool\WObj:=Workobject_1;
        MoveL Target_750,v100,z100,MyNewTool\WObj:=Workobject_1;
        MoveL Target_760,v100,z100,MyNewTool\WObj:=Workobject_1;
        MoveL Target_770,v100,z100,MyNewTool\WObj:=Workobject_1;
        MoveL Target_780,v100,z100,MyNewTool\WObj:=Workobject_1;
        MoveL Target_790,v100,z100,MyNewTool\WObj:=Workobject_1;
        MoveL Target_800,v100,z100,MyNewTool\WObj:=Workobject_1;
        MoveL Target_810,v100,z100,MyNewTool\WObj:=Workobject_1;
        MoveL Target_820,v100,z100,MyNewTool\WObj:=Workobject_1;
        MoveL Target_830,v100,z100,MyNewTool\WObj:=Workobject_1;
        MoveL Target_840_OExtFinal,v100,z100,MyNewTool\WObj:=Workobject_1;
        MoveL Target_730_OExtInicio,v100,z100,MyNewTool\WObj:=Workobject_1;
        MoveL Target_730_OExtInicio_2,v100,z100,MyNewTool\WObj:=Workobject_1;
    ENDPROC
    PROC Letra_OInt()
        MoveL Target_850_OIntInicio_3,v100,z100,MyNewTool\WObj:=Workobject_1;
        MoveL Target_850_OIntInicio,v100,z100,MyNewTool\WObj:=Workobject_1;
        MoveL Target_860,v100,z100,MyNewTool\WObj:=Workobject_1;
        MoveL Target_870,v100,z100,MyNewTool\WObj:=Workobject_1;
        MoveL Target_880,v100,z100,MyNewTool\WObj:=Workobject_1;
        MoveL Target_890,v100,z100,MyNewTool\WObj:=Workobject_1;
        MoveL Target_900,v100,z100,MyNewTool\WObj:=Workobject_1;
        MoveL Target_910,v100,z100,MyNewTool\WObj:=Workobject_1;
        MoveL Target_920,v100,z100,MyNewTool\WObj:=Workobject_1;
        MoveL Target_930,v100,z100,MyNewTool\WObj:=Workobject_1;
        MoveL Target_940,v100,z100,MyNewTool\WObj:=Workobject_1;
        MoveL Target_950,v100,z100,MyNewTool\WObj:=Workobject_1;
        MoveL Target_960_OIntFinal,v100,z100,MyNewTool\WObj:=Workobject_1;
        MoveL Target_850_OIntInicio,v100,z100,MyNewTool\WObj:=Workobject_1;
        MoveL Target_850_OIntInicio_3,v100,z100,MyNewTool\WObj:=Workobject_1;
    ENDPROC
    PROC Letra_K2()
        MoveL Target_970_K2Inicio_2,v100,z100,MyNewTool\WObj:=Workobject_1;
        MoveL Target_970_K2Inicio,v100,z100,MyNewTool\WObj:=Workobject_1;
        MoveL Target_980,v100,z100,MyNewTool\WObj:=Workobject_1;
        MoveL Target_990,v100,z100,MyNewTool\WObj:=Workobject_1;
        MoveL Target_1000,v100,z100,MyNewTool\WObj:=Workobject_1;
        MoveL Target_1010,v100,z100,MyNewTool\WObj:=Workobject_1;
        MoveL Target_1020,v100,z100,MyNewTool\WObj:=Workobject_1;
        MoveL Target_1030,v100,z100,MyNewTool\WObj:=Workobject_1;
        MoveL Target_1040,v100,z100,MyNewTool\WObj:=Workobject_1;
        MoveL Target_1050,v100,z100,MyNewTool\WObj:=Workobject_1;
        MoveL Target_1060,v100,z100,MyNewTool\WObj:=Workobject_1;
        MoveL Target_1070,v100,z100,MyNewTool\WObj:=Workobject_1;
        MoveL Target_1080_K2Final,v100,z100,MyNewTool\WObj:=Workobject_1;
        MoveL Target_970_K2Inicio,v100,z100,MyNewTool\WObj:=Workobject_1;
        MoveL Target_970_K2Inicio_2,v100,z100,MyNewTool\WObj:=Workobject_1;
    ENDPROC
    PROC Letra_C()
        MoveL Target_1090_CInicio_2,v100,z100,MyNewTool\WObj:=Workobject_1;
        MoveL Target_1090_CInicio,v100,z100,MyNewTool\WObj:=Workobject_1;
        MoveL Target_1100,v100,z100,MyNewTool\WObj:=Workobject_1;
        MoveL Target_1110,v100,z100,MyNewTool\WObj:=Workobject_1;
        MoveL Target_1120,v100,z100,MyNewTool\WObj:=Workobject_1;
        MoveL Target_1130,v100,z100,MyNewTool\WObj:=Workobject_1;
        MoveL Target_1140,v100,z100,MyNewTool\WObj:=Workobject_1;
        MoveL Target_1150,v100,z100,MyNewTool\WObj:=Workobject_1;
        MoveL Target_1160,v100,z100,MyNewTool\WObj:=Workobject_1;
        MoveL Target_1170,v100,z100,MyNewTool\WObj:=Workobject_1;
        MoveL Target_1180,v100,z100,MyNewTool\WObj:=Workobject_1;
        MoveL Target_1190,v100,z100,MyNewTool\WObj:=Workobject_1;
        MoveL Target_1200,v100,z100,MyNewTool\WObj:=Workobject_1;
        MoveL Target_1210,v100,z100,MyNewTool\WObj:=Workobject_1;
        MoveL Target_1220,v100,z100,MyNewTool\WObj:=Workobject_1;
        MoveL Target_1230,v100,z100,MyNewTool\WObj:=Workobject_1;
        MoveL Target_1240,v100,z100,MyNewTool\WObj:=Workobject_1;
        MoveL Target_1250,v100,z100,MyNewTool\WObj:=Workobject_1;
        MoveL Target_1260,v100,z100,MyNewTool\WObj:=Workobject_1;
        MoveL Target_1270,v100,z100,MyNewTool\WObj:=Workobject_1;
        MoveL Target_1280_CFinal,v100,z100,MyNewTool\WObj:=Workobject_1;
        MoveL Target_1090_CInicio,v100,z100,MyNewTool\WObj:=Workobject_1;
        MoveL Target_1090_CInicio_2,v100,z100,MyNewTool\WObj:=Workobject_1;
    ENDPROC
    PROC Letra_AExt()
        MoveL Target_1290_AExtInicio_2,v100,z100,MyNewTool\WObj:=Workobject_1;
        MoveL Target_1290_AExtInicio,v100,z100,MyNewTool\WObj:=Workobject_1;
        MoveL Target_1300,v100,z100,MyNewTool\WObj:=Workobject_1;
        MoveL Target_1310,v100,z100,MyNewTool\WObj:=Workobject_1;
        MoveL Target_1320,v100,z100,MyNewTool\WObj:=Workobject_1;
        MoveL Target_1330,v100,z100,MyNewTool\WObj:=Workobject_1;
        MoveL Target_1340,v100,z100,MyNewTool\WObj:=Workobject_1;
        MoveL Target_1350,v100,z100,MyNewTool\WObj:=Workobject_1;
        MoveL Target_1360_AExtFinal,v100,z100,MyNewTool\WObj:=Workobject_1;
        MoveL Target_1290_AExtInicio,v100,z100,MyNewTool\WObj:=Workobject_1;
        MoveL Target_1290_AExtInicio_2,v100,z100,MyNewTool\WObj:=Workobject_1;
    ENDPROC
    PROC Letra_J()
        MoveL Target_1400_JInicio_2,v100,z100,MyNewTool\WObj:=Workobject_1;
        MoveL Target_1400_JInicio,v100,z100,MyNewTool\WObj:=Workobject_1;
        MoveL Target_1410,v100,z100,MyNewTool\WObj:=Workobject_1;
        MoveL Target_1420,v100,z100,MyNewTool\WObj:=Workobject_1;
        MoveL Target_1430,v100,z100,MyNewTool\WObj:=Workobject_1;
        MoveL Target_1440,v100,z100,MyNewTool\WObj:=Workobject_1;
        MoveL Target_1450,v100,z100,MyNewTool\WObj:=Workobject_1;
        MoveL Target_1460,v100,z100,MyNewTool\WObj:=Workobject_1;
        MoveL Target_1470,v100,z100,MyNewTool\WObj:=Workobject_1;
        MoveL Target_1480,v100,z100,MyNewTool\WObj:=Workobject_1;
        MoveL Target_1490,v100,z100,MyNewTool\WObj:=Workobject_1;
        MoveL Target_1500_JFinal,v100,z100,MyNewTool\WObj:=Workobject_1;
        MoveL Target_1400_JInicio,v100,z100,MyNewTool\WObj:=Workobject_1;
        MoveL Target_1400_JInicio_2,v100,z100,MyNewTool\WObj:=Workobject_1;
    ENDPROC
    PROC Letra_T3()
        MoveL Target_1510_T3Inicio_2,v100,z100,MyNewTool\WObj:=Workobject_1;
        MoveL Target_1510_T3Inicio,v100,z100,MyNewTool\WObj:=Workobject_1;
        MoveL Target_1520,v100,z100,MyNewTool\WObj:=Workobject_1;
        MoveL Target_1530,v100,z100,MyNewTool\WObj:=Workobject_1;
        MoveL Target_1540,v100,z100,MyNewTool\WObj:=Workobject_1;
        MoveL Target_1550,v100,z100,MyNewTool\WObj:=Workobject_1;
        MoveL Target_1560,v100,z100,MyNewTool\WObj:=Workobject_1;
        MoveL Target_1570,v100,z100,MyNewTool\WObj:=Workobject_1;
        MoveL Target_1580_T3Final,v100,z100,MyNewTool\WObj:=Workobject_1;
        MoveL Target_1510_T3Inicio,v100,z100,MyNewTool\WObj:=Workobject_1;
        MoveL Target_1510_T3Inicio_2,v100,z100,MyNewTool\WObj:=Workobject_1;
    ENDPROC
    PROC Letra_AInt()
        MoveL Target_1370_AIntInicio_2,v100,z100,MyNewTool\WObj:=Workobject_1;
        MoveL Target_1370_AIntInicio,v100,z100,MyNewTool\WObj:=Workobject_1;
        MoveL Target_1380,v100,z100,MyNewTool\WObj:=Workobject_1;
        MoveL Target_1390_AIntFinal,v100,z100,MyNewTool\WObj:=Workobject_1;
        MoveL Target_1370_AIntInicio,v100,z100,MyNewTool\WObj:=Workobject_1;
        MoveL Target_1370_AIntInicio_2,v100,z100,MyNewTool\WObj:=Workobject_1;
    ENDPROC
    PROC Mantenimiento()
        MoveJ PosMantenimiento,v400,z100,MyNewTool\WObj:=Workobject_1;
    ENDPROC
    PROC Home()
        MoveJ MyHome,v400,z100,MyNewTool\WObj:=Workobject_1;
    ENDPROC
ENDMODULE
